FUNCTION_BLOCK FB2_Control
VAR_INPUT
END_VAR
VAR_OUTPUT
END_VAR
VAR
END_VAR

//loadingstation
Loadingstation.i_weighbridge.TruckOnScale 			:= Weighbridge.q_Output.TruckOnScale;
Loadingstation.i_weighbridge.WeightLimitReached 	:= Weighbridge.q_Output.WeightLimitReached;

Loadingstation(iq_Commandstate := GlobalCommandState);

END_FUNCTION_BLOCK

(* stored: Version 1.1.0.1, ProductVersion 3.1.4024.6
   POU FB2_Control: Id {f3ae371c-7e7d-41b3-b42c-11221479fa8f}, SpecialFunc None *)
